Yaskawa INFORM job: pos_z_0.JBI

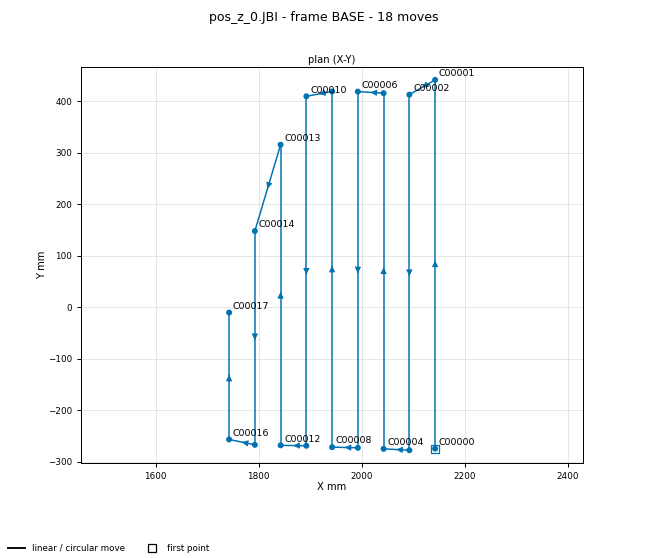
[picture p0: tool path of pos_z_0.JBI in frame BASE, 18 of 20 moves have a stored position in this frame; points joined in program order, loops and branches not executed]
/JOB
//NAME pos_z_0
//POS
///NPOS 18,0,18,0,0,0
///TOOL 0
///POSTYPE BASE
///RECTAN
///RCONF 0,0,0,0,0,0,0,0,0,0,0,0,0,0,0,0,0,0,0,0,0,0,0,0
C00000=2142.874513,-274.755902,-628.283050,175.000000,-5.000000,5.000000
C00001=2142.874513,441.314098,-629.348050,175.000000,-5.000000,5.000000
C00002=2092.874513,412.481098,-627.386050,175.000000,-5.000000,5.000000
C00003=2092.874513,-277.877902,-627.655050,175.000000,-5.000000,5.000000
C00004=2042.874513,-275.116902,-627.294050,175.000000,-5.000000,5.000000
C00005=2042.874513,415.422098,-627.433050,175.000000,-5.000000,5.000000
C00006=1992.874513,418.527098,-627.273050,175.000000,-5.000000,5.000000
C00007=1992.874513,-273.145902,-626.895050,175.000000,-5.000000,5.000000
C00008=1942.874513,-271.834902,-627.979050,175.000000,-5.000000,5.000000
C00009=1942.874513,418.747098,-627.591050,175.000000,-5.000000,5.000000
C00010=1892.874513,409.378098,-639.818050,175.000000,-5.000000,5.000000
C00011=1892.874513,-269.169902,-628.223050,175.000000,-5.000000,5.000000
C00012=1842.874513,-268.344902,-628.987050,175.000000,-5.000000,5.000000
C00013=1842.874513,315.419098,-629.428050,175.000000,-5.000000,5.000000
C00014=1792.874513,147.737098,-629.908050,175.000000,-5.000000,5.000000
C00015=1792.874513,-267.360902,-629.616050,175.000000,-5.000000,5.000000
C00016=1742.869513,-256.897902,-629.160050,175.000000,-5.000000,5.000000
C00017=1742.869513,-10.568602,-630.317050,175.000000,-5.000000,5.000000
///POSTYPE PULSE
///PULSE
EX000=0
///POSTYPE PULSE
///PULSE
EC00000=0
EC00001=0
EC00002=0
EC00003=0
EC00004=0
EC00005=0
EC00006=0
EC00007=0
EC00008=0
EC00009=0
EC00010=0
EC00011=0
EC00012=0
EC00013=0
EC00014=0
EC00015=0
EC00016=0
EC00017=0
//INST
///DATE 2023/08/07 14:38
///ATTR SC,RW,RJ
////FRAME BASE
///GROUP1 RB1,ST1
NOP
MOVJ P009 EX000 VJ=15.00
MOVJ C00000 EC00000 VJ=15.0
CALL JOB:SPYON
MOVL C00001 EC00001 V=150.0
MOVL C00002 EC00002 V=150.0
MOVL C00003 EC00003 V=150.0
MOVL C00004 EC00004 V=150.0
MOVL C00005 EC00005 V=150.0
MOVL C00006 EC00006 V=150.0
MOVL C00007 EC00007 V=150.0
MOVL C00008 EC00008 V=150.0
MOVL C00009 EC00009 V=150.0
MOVL C00010 EC00010 V=150.0
MOVL C00011 EC00011 V=150.0
MOVL C00012 EC00012 V=150.0
MOVL C00013 EC00013 V=150.0
MOVL C00014 EC00014 V=150.0
MOVL C00015 EC00015 V=150.0
MOVL C00016 EC00016 V=150.0
MOVL C00017 EC00017 V=150.0
CALL JOB:SPYOF
MOVJ P009 VJ=15.00
END
